FUNCTION_BLOCK FB_AlimentadorVerificadorDesplazador_SFC
VAR_INPUT
	//Tiempo
	Tcheck: TIME := T#1S;
	Tdesplazador: TIME := T#1S;
	
	// SFC-Flags
	SFCPause: BOOL;
	SFCReset: BOOL;
	
	//Indicadores de sincronizacion
	Ack: BOOL:= TRUE;
	Execute: BOOL;
	
	//Entradas
	
	Alimentador_delante: BOOL; //Bajo el verificador
	Alimentador_detras: BOOL;
	Verificador_arriba: BOOL;
	Verificador_abajo: BOOL;
	Desplazador_delante: BOOL;
	Desplazador_detras: BOOL;
	
END_VAR
VAR_OUTPUT
	//indicadores de sincronizacion
	Done: BOOL;
	Ready: BOOL;

	//Salidas
	Alimentador_adelante: BOOL;
	Verificador_baja: BOOL;
	Desplazador_adelante: BOOL;
	
	pieza_ok : BOOL;

END_VAR
VAR
END_VAR

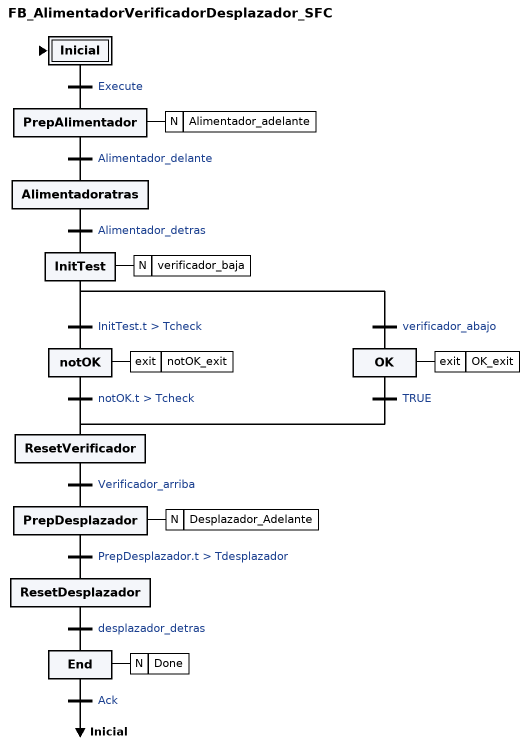
INITIAL_STEP Inicial:
END_STEP
TRANSITION FROM Inicial TO PrepAlimentador
    := Execute;
END_TRANSITION
STEP PrepAlimentador:
    Alimentador_adelante(N);
END_STEP
TRANSITION FROM PrepAlimentador TO Alimentadoratras
    := Alimentador_delante;
END_TRANSITION
STEP Alimentadoratras:
END_STEP
TRANSITION FROM Alimentadoratras TO InitTest
    := Alimentador_detras;
END_TRANSITION
STEP InitTest:
    verificador_baja(N);
END_STEP
TRANSITION FROM InitTest TO notOK
    := InitTest.t > Tcheck;
END_TRANSITION
STEP notOK:
    notOK_exit(P0);  // exit action
END_STEP
TRANSITION FROM notOK TO ResetVerificador
    := notOK.t > Tcheck;
END_TRANSITION
TRANSITION FROM InitTest TO OK
    := verificador_abajo;
END_TRANSITION
STEP OK:
    OK_exit(P0);  // exit action
END_STEP
TRANSITION FROM OK TO ResetVerificador
    := TRUE;
END_TRANSITION
STEP ResetVerificador:
END_STEP
TRANSITION FROM ResetVerificador TO PrepDesplazador
    := Verificador_arriba;
END_TRANSITION
STEP PrepDesplazador:
    Desplazador_Adelante(N);
END_STEP
TRANSITION FROM PrepDesplazador TO ResetDesplazador
    := PrepDesplazador.t > Tdesplazador;
END_TRANSITION
STEP ResetDesplazador:
END_STEP
TRANSITION FROM ResetDesplazador TO End
    := desplazador_detras;
END_TRANSITION
STEP End:
    Done(N);
END_STEP
TRANSITION FROM End TO Inicial
    := Ack;
END_TRANSITION

ACTION notOK_exit:
pieza_ok := FALSE;
END_ACTION

ACTION OK_exit:
pieza_ok := TRUE;
END_ACTION

END_FUNCTION_BLOCK

(* stored: Version 1.1.0.1, ProductVersion 3.1.4024.12
   POU FB_AlimentadorVerificadorDesplazador_SFC: Id {d0e02cd0-9cc1-42c8-afe4-bef33f1d13d0}, SpecialFunc None
   Action notOK_exit: Id {81cbfc81-a284-4b53-b11b-1cd41d253b6b}
   Action OK_exit: Id {7dd72752-0df9-435b-b4fe-3c9ac0cf4f73} *)
